TYPE ST_SHA256_BufferState :
STRUCT
	p				: PVOID;
	len				: UDINT;
	total			: UDINT;
	single_one_delivered	: BOOL;
	total_len_delivered		: BOOL;
END_STRUCT
END_TYPE

(* stored: Version 1.1.0.1, ProductVersion 3.1.4024.6
   DUT ST_SHA256_BufferState: Id {10b6f0bb-8d4e-4c6b-b966-b6da468fcb44} *)
